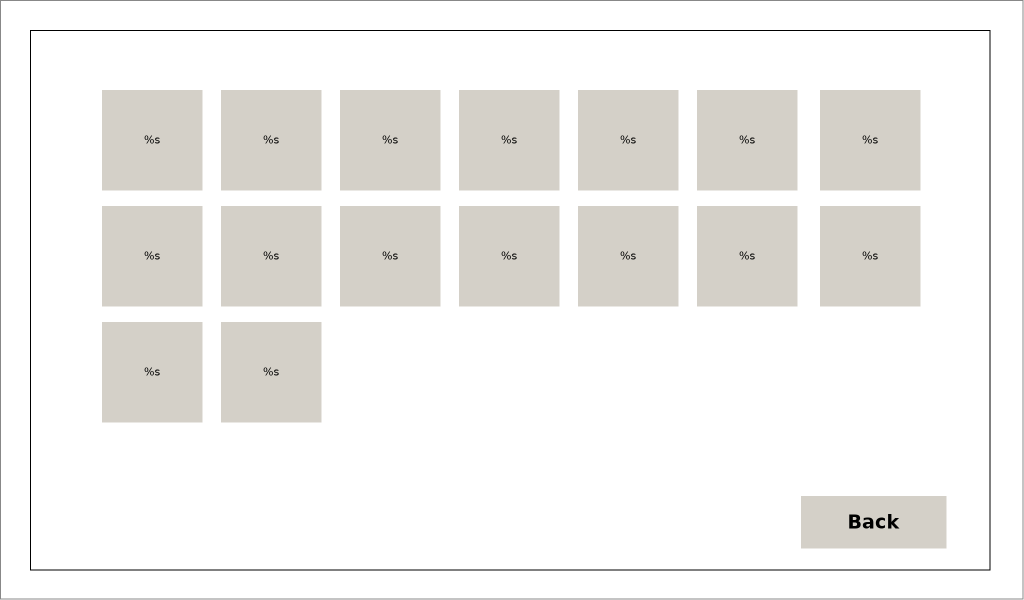
VISUALIZATION V_Builders  // 1024x600
VAR_IN_OUT
	HMI : ST_PackMLBaseModule_HMI;
	HMI_GantryXYZ : ST_GantryXYZ_HMI;
END_VAR
    RoundedRectangle (30,30 960x540)
    RoundedRectangle (801,496 145x52), "Back"
        OnMouseUp: execute { GVL_HMI.PopupToDisplay := 0; }
    RoundedRectangle (340,90 100x100), "%s", text variable: MAIN.Seedra.aRecipeNames[3], colour toggle: HMI_GantryXYZ.Command.ProgramIdRequested = 3, invisible if: MAIN.Seedra.aRecipeNames[3] = ''
        OnMouseClick: execute { HMI_GantryXYZ.Command.ProgramIdRequested := 3; }
        OnMouseUp: execute { GVL_HMI.PopupToDisplay := 0; }
    RoundedRectangle (221,90 100x100), "%s", text variable: MAIN.Seedra.aRecipeNames[2], colour toggle: HMI_GantryXYZ.Command.ProgramIdRequested = 2, invisible if: MAIN.Seedra.aRecipeNames[2] = ''
        OnMouseClick: execute { HMI_GantryXYZ.Command.ProgramIdRequested := 2; }
        OnMouseUp: execute { GVL_HMI.PopupToDisplay := 0; }
    RoundedRectangle (102,90 100x100), "%s", text variable: MAIN.Seedra.aRecipeNames[1], colour toggle: HMI_GantryXYZ.Command.ProgramIdRequested = 1, invisible if: MAIN.Seedra.aRecipeNames[1] = ''
        OnMouseClick: execute { HMI_GantryXYZ.Command.ProgramIdRequested := 1; }
        OnMouseUp: execute { GVL_HMI.PopupToDisplay := 0; }
    RoundedRectangle (459,90 100x100), "%s", text variable: MAIN.Seedra.aRecipeNames[4], colour toggle: HMI_GantryXYZ.Command.ProgramIdRequested = 4, invisible if: MAIN.Seedra.aRecipeNames[4] = ''
        OnMouseClick: execute { HMI_GantryXYZ.Command.ProgramIdRequested := 4; }
        OnMouseUp: execute { GVL_HMI.PopupToDisplay := 0; }
    RoundedRectangle (578,90 100x100), "%s", text variable: MAIN.Seedra.aRecipeNames[5], colour toggle: HMI_GantryXYZ.Command.ProgramIdRequested = 5, invisible if: MAIN.Seedra.aRecipeNames[5] = ''
        OnMouseClick: execute { HMI_GantryXYZ.Command.ProgramIdRequested := 5; }
        OnMouseUp: execute { GVL_HMI.PopupToDisplay := 0; }
    RoundedRectangle (697,90 100x100), "%s", text variable: MAIN.Seedra.aRecipeNames[6], colour toggle: HMI_GantryXYZ.Command.ProgramIdRequested = 6, invisible if: MAIN.Seedra.aRecipeNames[6] = ''
        OnMouseClick: execute { HMI_GantryXYZ.Command.ProgramIdRequested := 6; }
        OnMouseUp: execute { GVL_HMI.PopupToDisplay := 0; }
    RoundedRectangle (820,90 100x100), "%s", text variable: MAIN.Seedra.aRecipeNames[7], colour toggle: HMI_GantryXYZ.Command.ProgramIdRequested = 7, invisible if: MAIN.Seedra.aRecipeNames[7] = ''
        OnMouseClick: execute { HMI_GantryXYZ.Command.ProgramIdRequested := 7; }
        OnMouseUp: execute { GVL_HMI.PopupToDisplay := 0; }
    RoundedRectangle (102,206 100x100), "%s", text variable: MAIN.Seedra.aRecipeNames[8], colour toggle: HMI_GantryXYZ.Command.ProgramIdRequested = 8, invisible if: MAIN.Seedra.aRecipeNames[8] = ''
        OnMouseClick: execute { HMI_GantryXYZ.Command.ProgramIdRequested := 8; }
        OnMouseUp: execute { GVL_HMI.PopupToDisplay := 0; }
    RoundedRectangle (221,206 100x100), "%s", text variable: MAIN.Seedra.aRecipeNames[9], colour toggle: HMI_GantryXYZ.Command.ProgramIdRequested =9, invisible if: MAIN.Seedra.aRecipeNames[9] = ''
        OnMouseClick: execute { HMI_GantryXYZ.Command.ProgramIdRequested := 9; }
        OnMouseUp: execute { GVL_HMI.PopupToDisplay := 0; }
    RoundedRectangle (340,206 100x100), "%s", text variable: MAIN.Seedra.aRecipeNames[10], colour toggle: HMI_GantryXYZ.Command.ProgramIdRequested = 10, invisible if: MAIN.Seedra.aRecipeNames[10] = ''
        OnMouseClick: execute { HMI_GantryXYZ.Command.ProgramIdRequested := 10; }
        OnMouseUp: execute { GVL_HMI.PopupToDisplay := 0; }
    RoundedRectangle (459,206 100x100), "%s", text variable: MAIN.Seedra.aRecipeNames[11], colour toggle: HMI_GantryXYZ.Command.ProgramIdRequested = 11, invisible if: MAIN.Seedra.aRecipeNames[11] = ''
        OnMouseClick: execute { HMI_GantryXYZ.Command.ProgramIdRequested := 11; }
        OnMouseUp: execute { GVL_HMI.PopupToDisplay := 0; }
    RoundedRectangle (578,206 100x100), "%s", text variable: MAIN.Seedra.aRecipeNames[12], colour toggle: HMI_GantryXYZ.Command.ProgramIdRequested = 12, invisible if: MAIN.Seedra.aRecipeNames[12] = ''
        OnMouseClick: execute { HMI_GantryXYZ.Command.ProgramIdRequested := 12; }
        OnMouseUp: execute { GVL_HMI.PopupToDisplay := 0; }
    RoundedRectangle (697,206 100x100), "%s", text variable: MAIN.Seedra.aRecipeNames[13], colour toggle: HMI_GantryXYZ.Command.ProgramIdRequested = 13, invisible if: MAIN.Seedra.aRecipeNames[13] = ''
        OnMouseClick: execute { HMI_GantryXYZ.Command.ProgramIdRequested := 13; }
        OnMouseUp: execute { GVL_HMI.PopupToDisplay := 0; }
    RoundedRectangle (820,206 100x100), "%s", text variable: MAIN.Seedra.aRecipeNames[14], colour toggle: HMI_GantryXYZ.Command.ProgramIdRequested = 14, invisible if: MAIN.Seedra.aRecipeNames[14] = ''
        OnMouseClick: execute { HMI_GantryXYZ.Command.ProgramIdRequested := 14; }
        OnMouseUp: execute { GVL_HMI.PopupToDisplay := 0; }
    RoundedRectangle (102,322 100x100), "%s", text variable: MAIN.Seedra.aRecipeNames[15], colour toggle: HMI_GantryXYZ.Command.ProgramIdRequested = 15, invisible if: MAIN.Seedra.aRecipeNames[15] = ''
        OnMouseClick: execute { HMI_GantryXYZ.Command.ProgramIdRequested := 15; }
        OnMouseUp: execute { GVL_HMI.PopupToDisplay := 0; }
    RoundedRectangle (221,322 100x100), "%s", text variable: MAIN.Seedra.aRecipeNames[16], colour toggle: HMI_GantryXYZ.Command.ProgramIdRequested = 16, invisible if: MAIN.Seedra.aRecipeNames[16] = ''
        OnMouseClick: execute { HMI_GantryXYZ.Command.ProgramIdRequested := 16; }
        OnMouseUp: execute { GVL_HMI.PopupToDisplay := 0; }
END_VISUALIZATION

(* stored: Version 1.1.0.1, ProductVersion 3.1.4024.15
   Visu V_Builders: Id {58acf0c6-591c-4396-a407-7b3fb6febf1a} *)
